FUNCTION F_Log : BOOL
VAR_INPUT
	fbMessage:			REFERENCE TO FB_Message;
END_VAR
VAR
	sMessage:			STRING(255):= 'Logger null | ';
    nIndex:				UINT;
    nNow:				ULINT:= F_GetSystemTime();
END_VAR


// --- Build log line
sMessage := CONCAT('Logger null | ', fbMessage.sSource);
sMessage := CONCAT(sMessage, ': ');
sMessage := CONCAT(sMessage, fbMessage.sDefault);

// --- Keep active
nIndex := 0;
WHILE nIndex < nBuffer DO
    IF aBuffer[nIndex].sDefault = fbMessage.sDefault THEN
		aBuffer[nIndex].bActive:= TRUE;
        F_Log := TRUE;
        RETURN;
    END_IF
    nIndex := nIndex + 1;
END_WHILE

// --- Add to buffer ---
IF nBuffer < UPPER_BOUND(aBuffer, 1) THEN
    aBuffer[nBuffer] := fbMessage;
    aBuffer[nBuffer].nTimestamp := nNow;
    nBuffer := nBuffer + 1;
END_IF

// --- Log message ---
CASE fbMessage.eLogLevel OF
    E_LogLevel.Verbose, E_LogLevel.Info:
        ADSLOGSTR(ADSLOG_MSGTYPE_HINT, '%s', sMessage);
    E_LogLevel.Warning:
        ADSLOGSTR(ADSLOG_MSGTYPE_WARN, '%s', sMessage);
    E_LogLevel.Error, E_LogLevel.Critical:
        ADSLOGSTR(ADSLOG_MSGTYPE_ERROR, '%s', sMessage);
END_CASE

// --- Remove outdated messages (>1 s old) ---
nIndex := 0;
WHILE nIndex < nBuffer DO
    IF (nNow - aBuffer[nIndex].nTimestamp) > 1_000_000_000 THEN // 1 s = 1e9 ns
        MEMMOVE(ADR(aBuffer[nIndex]), ADR(aBuffer[nIndex + 1]), SIZEOF(FB_Message) * (nBuffer - nIndex - 1));
        nBuffer := nBuffer - 1;
    ELSE
        nIndex := nIndex + 1;
    END_IF
END_WHILE


F_Log := TRUE;

END_FUNCTION

(* stored: Version 1.1.0.1
   POU F_Log: Id {3d8b8d8d-2aeb-485f-a382-76004536aaec}, SpecialFunc None *)
